// TIA Portal V18 export
FUNCTION_BLOCK "SysFlowCtrlGraph"   // FB3006, SCL
{ S7_Optimized_Access := 'TRUE' }
VERSION : 0.1
// stored: AutoNumber false, IsIECCheckEnabled false, IsRetainMemResEnabled false, MemoryReserve 100, SetENOAutomatically false, UDAEnableTagReadback false
   VAR_INPUT
      iSysInface : "RCS_SysComInterface_V1";
   END_VAR
   VAR_IN_OUT
      ioPM_Inface : "RCS_PMInterface_V1";
      ioGraphCtrl : G7_MOPPlus_V6;
   END_VAR
   VAR
      sHis : Array[0..7] of Bool;
      sSetInitialDelay : TON_TIME;
      S_NEXT_Delay { S7_SetPoint := 'True'} : Array[0..1] of TON_TIME;
   END_VAR
BEGIN
   (*############################################################
      RUHLAMAT SUZHOU ELEC.STD.
      Copyright (c) 2022. All rights reserved.    

      NAME OF FUNCTION BLOCK:         SysFlowCtrlGraph
      VERSION NUMBER:                 V1.0
      COMPOSER:                       Ming.Jiang

      LAST CHANGE:                    1.Dece.2022
      Comment by Ming.Jiang 

      #RET_VALUE:


      #Alert Value:


      -----------------------------------------------------
      Date        Name      Version           Activity                                                                              

   ############################################################*)

   REGION Control Mode
       //AUTO:Auto Mode
       #ioGraphCtrl.AUTO := #ioGraphCtrl.SUP := #iSysInface.Auto.Mode;

       //MAN:Manual Mode
       #ioGraphCtrl.MAN :=  #iSysInface.ManualMode;
       #ioGraphCtrl.OFF := #ioPM_Inface.AlarmImdilyStop OR #iSysInface.ManualMode;
       IF #iSysInface.ManualMode OR #ioPM_Inface.AlarmImdilyStop THEN
           #ioPM_Inface.InitialRun      := 0;
           #ioPM_Inface.InitialOK       := 0;
           #ioPM_Inface.WaitRunning     := 0;
           // #ioPM_Inface.Running         := 0;
           #ioPM_Inface.UnPause    := 0;
           #ioPM_Inface.ProcessComplete := 0;

       END_IF;
       //AutoRunning
       //
       // #ioPM_Inface.Running := ((#iSysInface.Auto.StartAuto AND #iSysInface.Ready) OR #iSysInface.Auto.Running)
       // AND AND NOT "ST10_Sys".Auto.RunningOver 

       IF NOT #iSysInface.ManualMode AND #iSysInface.SysRun AND #ioPM_Inface.InitialOK AND NOT #ioPM_Inface.Alarm
           AND NOT #ioPM_Inface.AlarmImdilyStop AND NOT #iSysInface.Auto.RunningPause THEN
           IF #iSysInface.Auto.StartAuto AND #iSysInface.Ready AND  NOT  #ioPM_Inface.Running  THEN
               #ioPM_Inface.Running := 1;
           END_IF;
       ELSE
           #ioPM_Inface.Running := 0;
       END_IF;

       //Step Num






       //TAP:StepMode
       #ioGraphCtrl.TAP := #iSysInface.Auto.StepMode;
       #ioGraphCtrl.T_PUSH := #iSysInface.Auto.StepMode AND #ioPM_Inface.SetNextStep AND NOT #sHis[0];
       #sHis[0] := #ioPM_Inface.SetNextStep;

       //INTERLOCK
       #ioGraphCtrl.LOCK    := 1;
       #ioGraphCtrl.IL_PERM := 1;
       #ioGraphCtrl.T_PERM  := 1;

   END_REGION

   REGION Initialization

       #sSetInitialDelay(IN := #iSysInface.SetInitial OR #ioPM_Inface.SetInitial,
                         PT := T#2000ms);//20221221DB

       IF #sSetInitialDelay.Q AND #iSysInface.SysRun AND NOT #iSysInface.ManualMode THEN

           IF NOT #sHis[1] THEN
               //     #oStatus.Initializing := TRUE;
               //     #oStatus.InitializeOK := 0;
               //     #oStatus.WaitRunning := 0;
               //     #oStatus.Running := 0;
               //     #oStatus.RunningPause := 0;
               //     #oStatus.RunningFinished := 0;
               #ioGraphCtrl.INIT := #sSetInitialDelay.Q;
           END_IF;

       ELSE
           #ioGraphCtrl.INIT := 0;
       END_IF;
       #sHis[1] := #sSetInitialDelay.Q;
   END_REGION

   REGION Reset
       //
       #ioGraphCtrl.ACK := #iSysInface.Reset;


   END_REGION

   REGION Running and Pause(Halt)
       #ioGraphCtrl.HALT :=(#ioPM_Inface.InitialOK AND NOT #ioPM_Inface.Running )  OR   #ioPM_Inface.Alarm OR #ioPM_Inface.AlarmImdilyStop ; //#ioPM_Inface.UnPause  NOT #iSysInface.Auto.RunningPause
       #ioGraphCtrl.OPS_ZERO := #iSysInface.ManualMode OR NOT #iSysInface.SysRun OR #ioPM_Inface.AlarmImdilyStop ;
       #ioGraphCtrl.TMS_HALT := #iSysInface.ManualMode OR NOT #iSysInface.SysRun OR #ioPM_Inface.AlarmImdilyStop;
   END_REGION


   #S_NEXT_Delay[0](PT := t#3s,
                 IN := #ioGraphCtrl.S_NEXT);

   IF #S_NEXT_Delay[0].Q THEN
       #ioGraphCtrl.S_NEXT := 0;

   END_IF;

   #S_NEXT_Delay[1](PT := t#3s,
                    IN := NOT #ioGraphCtrl.S_NEXT);

   IF #S_NEXT_Delay[1].Q THEN
       #ioGraphCtrl.S_NEXT := 1;
   END_IF;
END_FUNCTION_BLOCK
